# EPICS autosave request: tests/testfiles/cfg/SF_DCOL_PV.req
$(SYS):GAP
$(SYS):CENTER
